{attribute 'GeneratedUsingTerminal: EL6861-0000-0016'}
{attribute addProperty BoxType "EL6861-0000-0016"}
{attribute addProperty Id "StatusAT %I*Status_7BCA2D079Data_InAT %I*ARRAY[0..127] OF USINT128"}
{attribute addProperty CRC "2401738004"}
{attribute addProperty Size "137"}
TYPE COM_TxPDO_Map_Inputs_93BAD1D7 :
STRUCT
	{attribute addProperty Name "Status"}
	Status AT %I* : Status_7BCA2D07;
	{attribute addProperty Name "Data_In"}
	Data_In AT %I* : ARRAY[0..127] OF USINT;
END_STRUCT
END_TYPE

(* stored: Version 1.2.0.0, ProductVersion 3.1.4024.9
   DUT COM_TxPDO_Map_Inputs_93BAD1D7: Id {0aaf8929-16fd-44f5-b5ec-a2e6a1e173a0} *)
